// TIA Portal V19 export
FUNCTION "SAMPLE_FUNCTION" : Void   // FC1, LAD
TITLE = SAMPLE FUNCTION FOR TESTING DOCUMENTATION
{ S7_Optimized_Access := 'TRUE' }
// stored: SetENOAutomatically false
   VAR_TEMP
      Start : Bool;   // Start Command
      Stop : Bool;   // Stop Command
      Running : Bool;   // Running ? (Y/N)
   END_VAR
BEGIN

REGION Network 1: Basic Latching Function
   // This is A Comment to Test The Documentation Prints Correctly
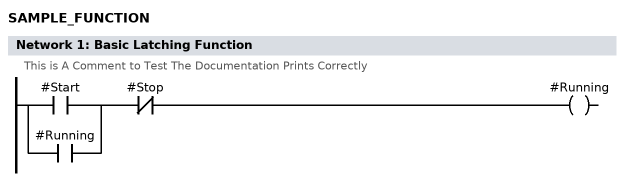
   RUNG wire#powerrail
      Contact( #Start )
      wire#w1
      I_Contact( #Stop )
      Coil( #Running )
   END_RUNG
   RUNG wire#powerrail
      Contact( #Running )
   END_RUNG wire#w1
   // the same network as SCL:
   #Running := (#Start OR #Running) AND NOT #Stop;
END_REGION
END_FUNCTION
